FUNCTION_BLOCK FB_PID_ROC
VAR_INPUT
	DisableROC			: BOOL;
	ValueIn				: REAL;
	LLM					: REAL; (* Setpoint low limit	*)
	HLM					: REAL; (* Setpoint high limit	*)
	ROC_UP				: REAL;
	ROC_DN				: REAL;
	tTskCycleTime		: TIME;
END_VAR
VAR_OUTPUT
	ValueOut			: REAL;
END_VAR
VAR
	OldValueIN			: REAL;
	ROC_UpLimit			: BOOL;
	ROC_DownLimit			: BOOL;
	CycleTimeSeconds	: REAL;
	ROC_UP_PerCycle		: REAL;
	ROC_DN_PerCycle		: REAL;
END_VAR
VAR // added by the converter: edge detectors and wires of the graphical bodies
    _w1, _w2 : BOOL;
END_VAR

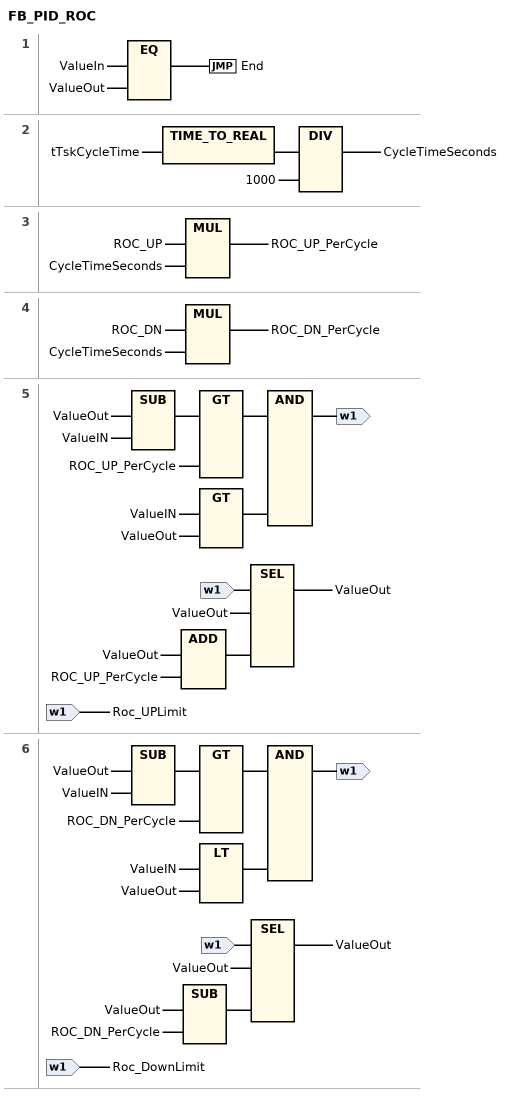
// NETWORK 1
IF ValueIn = ValueOut THEN JMP End; END_IF

// NETWORK 2
CycleTimeSeconds := TIME_TO_REAL(tTskCycleTime) / 1000;

// NETWORK 3
ROC_UP_PerCycle := ROC_UP * CycleTimeSeconds;

// NETWORK 4
ROC_DN_PerCycle := ROC_DN * CycleTimeSeconds;

// NETWORK 5
_w1 := ValueOut - ValueIN > ROC_UP_PerCycle AND ValueIN > ValueOut;
ValueOut := SEL(_w1, ValueOut, ValueOut + ROC_UP_PerCycle);
Roc_UPLimit := _w1;

// NETWORK 6
_w2 := ValueOut - ValueIN > ROC_DN_PerCycle AND ValueIN < ValueOut;
ValueOut := SEL(_w2, ValueOut, ValueOut - ROC_DN_PerCycle);
Roc_DownLimit := _w2;

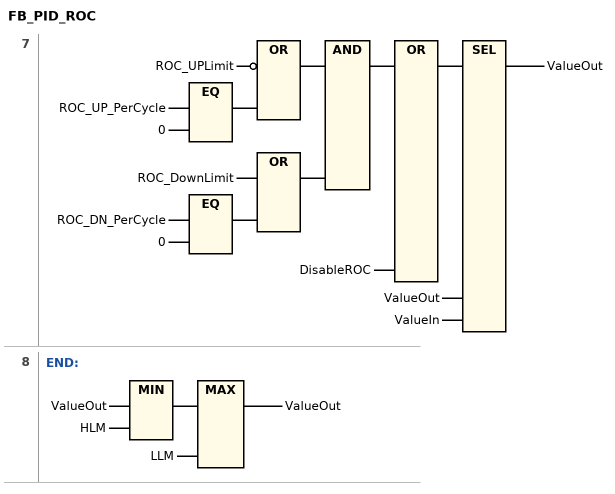
// NETWORK 7
ValueOut := SEL((NOT ROC_UPLimit OR ROC_UP_PerCycle = 0) AND (ROC_DownLimit OR ROC_DN_PerCycle = 0) OR DisableROC, ValueOut, ValueIn);

// NETWORK 8
END:
ValueOut := MAX(MIN(ValueOut, HLM), LLM);

END_FUNCTION_BLOCK

(* stored: Version 1.1.0.1, ProductVersion 3.1.4020.12
   POU FB_PID_ROC: Id {c98d3a7f-5b4d-4992-8d79-00828f784bd7}, SpecialFunc None *)
